Staubli VAL3: onF1Event.pgx

program onF1Event()
  local num l_nJogVelocity
  local num l_nSpeedScale
begin
  // look if the bButton is enable
  if bButton[0]
    // decrease the move


    ////    io:direction_neg=true
    ////    wait(getKey()==-1)
    ////    io:direction_neg=false


//    if ! isPowered()
//       call use:timerDialog("请给手臂上电",1)
//      return
//    endIf

    if aioGet(MbAI_bMotorPowe)==1
      ////7轴负向移动速度
      l_nJogVelocity=100
      ////
      aioSet(MbAO_aJogVelo,l_nJogVelocity)
      aioSet(MbAO_bMoveDirM,1)
      aioSet(MbAO_b7Axis,1)
      call use:timerDialog("7轴负向移动...",0)
    else
      if aioGet(MbAI_bMotorPowe)==0
        call use:timerDialog("7轴未上电",1)
        return
      endIf
    endIf


  endIf
  //

end
